FUNCTION_BLOCK T_ClearGroupCountEqualsZeroCompareEqualsFalse EXTENDS T_UnitTestBase
VAR
  list : T_ComponentsCollection;
  newComponent : ARRAY [1..5] OF T_ComponentMock;
  afterCountActual, afterCountExpected : UDINT;
  beforeCountActual, beforeCountExpected : UDINT;
  beforeActual, beforeExpected : I_ComponentBase;
  afterActual, afterExpected : I_ComponentBase;
 beforeResult, afterResult : BOOL;
END_VAR

// Arrange
list.AddComponent(newComponent[1]);
list.AddComponent(newComponent[2]);
list.AddComponent(newComponent[3]);
list.AddComponent(newComponent[4]);

// first test before running clear
beforeExpected := newComponent[1];
list.TryGetComponent(0, component => beforeActual);
beforeResult := beforeExpected = beforeActual;

Assertion.AssertEquals_BOOL(TRUE, beforeResult, 'item 0 = list.AddComponent()');
Assertion.AssertEquals_UDINT(4, list.Count, 'list.Count = 4');

//Act
list.ClearGroup();

//Assert 
afterExpected := newComponent[1];
list.TryGetComponent(0, component => afterActual);
afterResult := afterExpected <> afterActual;
Assertion.AssertEquals_BOOL(TRUE, beforeResult, 'afterResult := afterExpected <> afterActual;');

afterCountActual := list.Count;
afterCountExpected := 0;
Assertion.AssertEquals_UDINT(afterCountExpected, afterCountActual, 'afterCountActul = 0');

TestFinished();

END_FUNCTION_BLOCK

(* stored: Version 1.1.0.1, ProductVersion 3.1.4024.12
   POU T_ClearGroupCountEqualsZeroCompareEqualsFalse: Id {a5ac6aae-d815-4031-8abd-dd6bd35c8542}, SpecialFunc None *)
